// :Description: Rolling-average filter (library code under test).
FUNCTION_BLOCK FB_Filter
VAR_INPUT
    input : LREAL;
END_VAR
VAR_OUTPUT
    output : LREAL;
END_VAR
VAR
    state : E_State := E_State.Idle;
END_VAR


output := input;


// :Description: Advance the filter by one sample.
METHOD Step : LREAL
VAR_INPUT
    sample : LREAL;
END_VAR

Step := sample;
END_METHOD

END_FUNCTION_BLOCK

(* stored: Version 1.1.0.1, ProductVersion 3.1.4026.0
   POU FB_Filter: Id {aaaaaaaa-aaaa-aaaa-aaaa-aaaaaaaaaaa1}, SpecialFunc None
   Method Step: Id {aaaaaaaa-aaaa-aaaa-aaaa-aaaaaaaaaaa2} *)
